# EPICS StreamDevice protocol: proto/keithley.proto
OutTerminator = CR LF;
InTerminator = CR LF;
ReplyTimeout = 60000;

get_fields {
  Separator = ',';
  extrainput = ignore;
  replyTimeout = 1000;
  out "FETCH?";
  in "%f";
}
get_tracedata {
  Separator = ',';
  extrainput = ignore;
  replyTimeout = 1000;
  out ":TRAC:DATA?";
  in "%f";
}

sendtxt {
  out "%s";
}

disp {
  out ":DISP:ENAB %s";
  in  ":DISP:ENAB?";
}

cmd {
  out "\$1";
}

setVar {
  out "\$1 %f";
  @init {
    out "\$1?";
    in  "%f";
  }
}
getVar {
  out "\$1?";
  in  "%f";
}

setIntVar {
  out "\$1 %d";
  @init {
    out "\$1?";
    in  "%d";
  }
}
getIntVar {
  out "\$1?";
  in  "%d";
}

#setOffOn {
#  out "\$1 %{OFF|ON}";
#  @init {
#    out "\$1?";
#    in "%{0|1}";
#  }
#}
#getOffOn {
#  out "\$1??";
#  in "%{0|1}";
#}

getLSI {
  out "\$1";
  in  "%#s";
  ExtraInput = Ignore;
}

setDig {
  out ":SENS:VOLT:DIG %{8|7|6|5|4}";
  @init {
    out ":SENS:VOLT:DIG?";
    in  "%{8|7|6|5|4}";
  }
}
getDig {
  out ":SENS:VOLT:DIG?";
  in  "%{8|7|6|5|4}";
}

fetchTraceData {
  ReplyTimeout = 60000;
  Separator = ',';
  ExtraInput = Ignore;
  out ":TRAC:DATA?";
  in "%f";
}

setTrigSrc {
  out ":TRIG:SOURCE %{IMM|EXT}";
  @init {
    out ":TRIG:SOURCE?";
    in  "%{IMM|EXT}";
  }
}
getTrigSrc {
  out ":TRIG:SOURCE?";
  in  "%{IMM|EXT}";
}

setFeedCon {
  extrainput = ignore;
  out ":TRAC:FEED:CONT %{NEXT|NEVER}";
  @init {
    out ":TRAC:FEED:CONT?";
    in  "%{NEXT|NEV}";
  }
}
getFeedCon {
  extrainput = ignore;
  out ":TRAC:FEED:CONT?";
  in  "%{NEXT|NEV}";
}

setFeed {
  extrainput = ignore;
  out ":TRAC:FEED %{NONE|SENS|CALC}";
  @init {
    out ":TRAC:FEED?";
    in  "%{NONE|SENS|CALC}";
  }
}
getFeed {
  extrainput = ignore;
  out ":TRAC:FEED?";
  in  "%{NONE|SENS|CALC}";
}

setChan {
  out ":SENS:CHAN %{1|2}";
  @init {
    out ":SENS:CHAN?";
    in  "%{1|2}"
  }
}
getChan {
  out ":SENS:CHAN?";
  in  "%{1|2}"
}

setFunc {
  out ":SENS:FUNC \'%{VOLT:DC|TEMP}\'";
  @init {
    out ":SENS:FUNC?";
    in "%{\"VOLT:DC\"|\"TEMP\"}";
  }
}
getFunc {
  out ":SENS:FUNC?";
  in "%{\"VOLT:DC\"|\"TEMP\"}";
}

setRange {
  out ":SENS:VOLT:CHAN1:RANG %{0.010000|0.100000|1.000000|10.000000|100.000000}";
  @init {
    out ":SENS:VOLT:CHAN1:RANG?";
    in "%{0.010000|0.100000|1.000000|10.000000|100.000000}";
  }
}
getRange {
  out ":SENS:VOLT:CHAN1:RANG?";
  in "%{0.010000|0.100000|1.000000|10.000000|100.000000}";
  ExtraInput = Ignore;
}
